{attribute addProperty BoxType "EK1122-0000-0018"}
{attribute addProperty Id "Beckhoff_EP9xxxsub_EK1100EK1100_179A0949162A_0001_EP9128_0020_0016A_0001_EP9128_0020_0016_8825F3594744593"}
{attribute addProperty CRC "2290881861"}
{attribute addProperty SizeInBites "4760"}
{attribute addProperty SizeInBytes "595"}
TYPE Beckhoff_EP9xxxEK1122_888C1545 EXTENDS EK1122_179A0949 :
STRUCT
	{attribute addProperty Name "Beckhoff_EP9xxxsub_EK1100"}
	Beckhoff_EP9xxxsub_EK1100 : EK1100_179A0949;
	{attribute addProperty Name "A_0001_EP9128_0020_0016"}
	A_0001_EP9128_0020_0016 : A_0001_EP9128_0020_0016_8825F359;
END_STRUCT
END_TYPE

(* stored: Version 1.2.0.0, ProductVersion 3.1.4024.9
   DUT Beckhoff_EP9xxxEK1122_888C1545: Id {06f6b4a0-b3d0-4627-82a5-f9625aa28dfa} *)
